FUNCTION_BLOCK SERVERW (* Server for newline-terminated double-byte strings *)
  (* Standard: 61499-1 *)
  (* Version 0.0, 2004-10-15, JHC, Rockwell Automation *)
  (* Compiler header: package fb.rt.net; *)
  (* Compiler Java Sun JDK 1.4.2 *)
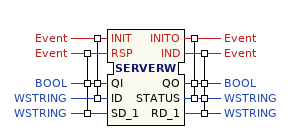
  EVENT_INPUT
    INIT WITH QI, ID;
    RSP WITH SD_1, QI; (* Response from server *)
  END_EVENT
  EVENT_OUTPUT
    INITO WITH QO, STATUS;
    IND WITH STATUS, QO, RD_1; (* Request to server *)
  END_EVENT
  VAR_INPUT
    QI : BOOL;
    ID : WSTRING; (* IP Socket Address *)
    SD_1 : WSTRING; (* String to be sent with added newline *)
  END_VAR
  VAR_OUTPUT
    QO : BOOL;
    STATUS : WSTRING;
    RD_1 : WSTRING; (* Received String without terminating newline *)
  END_VAR
END_FUNCTION_BLOCK
